// TIA Portal V17 export
// export: Created 2026-07-18T06:00:00.0000000Z, ExportSetting WithDefaults
DATA_BLOCK "GlobalData"   // DB1
{ S7_Optimized_Access := 'TRUE' }
VERSION : 0.1
// stored: AutoNumber true, IsIECCheckEnabled false
   VAR
      Ready : Bool;
      Count : Int;
      Config : Struct
         MaxSpeed : Real;
         Enabled : Bool;
      END_STRUCT;
   END_VAR
BEGIN
END_DATA_BLOCK
